// TIA Portal project "PaintMixingPlant" (V15)

(* hardware
DEVICE "S7-1200 station_1"  S7-1200 Station
   slot 0: "Rack_0"  S7-1200 Rack  Rack  V1.0
   slot 1: "PLC_1"  CPU 1214C AC/DC/Rly  6ES7 214-1BG40-0XB0  V4.2
DEVICE "PC-System_1"  SIMATIC PC station
   slot 0: "SIMATIC PC station"  Rail  SIMATIC PC-Station  V1.0
      slot 125: "Stationmanager"  Station_Manager  V6.0.4
   slot 1: "HMI_RT_1"  WinCC RT Professional  6AV2 105-0xxxx-xxxx  15.0.0.0
   slot 2: "IE general_1"  IE General  IE_CP  V8.2.0
*)

// ===== PLC "PLC_1"  CPU 1214C AC/DC/Rly =====

VAR_GLOBAL   // PLC tag table "Default tag table"
   "Mix1Tank1" AT %MW0 : Int;
   "Mix1Tank2" AT %MW2 : Int;
   "Mix1Tank3" AT %MW4 : Int;
   "Mix2Tank1" AT %MW6 : Int;
   "Mix2Tank2" AT %MW8 : Int;
   "Mix2Tank3" AT %MW10 : Int;
   "Mix3Tank1" AT %MW12 : Int;
   "Mix3Tank2" AT %MW14 : Int;
   "Mix3Tank3" AT %MW16 : Int;
   "InitM1T1" AT %MW18 : Int;
   "InitM1T2" AT %MW20 : Int;
   "InitM1T3" AT %MW22 : Int;
   "InitM2T1" AT %MW24 : Int;
   "InitM2T2" AT %MW26 : Int;
   "InitM2T3" AT %MW28 : Int;
   "InitM3T1" AT %MW30 : Int;
   "InitM3T2" AT %MW32 : Int;
   "InitM3T3" AT %MW34 : Int;
   "Tank1In" AT %MW36 : Int;
   "Tank1Out" AT %MW38 : Int;
   "Tank2In" AT %MW40 : Int;
   "Tank2Out" AT %MW42 : Int;
   "Tank3In" AT %MW44 : Int;
   "Tank3Out" AT %MW46 : Int;
   "Batch1In" AT %MW48 : Int;
   "Batch1Out" AT %MW50 : Int;
   "Batch2In" AT %MW52 : Int;
   "Batch2Out" AT %MW54 : Int;
   "Batch3In" AT %MW56 : Int;
   "Batch3Out" AT %MW58 : Int;
   "MixerIn" AT %MW60 : Int;
   "MixerOut" AT %MW62 : Int;
   "Start_Pb" AT %M64.0 : Bool;
   "Start_Trigger" AT %M64.1 : Bool;
   "Start" AT %M64.2 : Bool;
   "Stop_Pb" AT %M64.3 : Bool;
   "Stop_Trigger" AT %M64.4 : Bool;
   "InitStart" AT %M64.5 : Bool;
   "NextMix" AT %M64.6 : Bool;
   "ResetInd" AT %M64.7 : Bool;
   "Current_Mix" AT %MW66 : Int;
   "NumberOfMix1" AT %MW68 : Int;
   "Mix1Reset" AT %M65.0 : Bool;
   "NumberOfMix2" AT %MW70 : Int;
   "Mix2Reset" AT %M65.1 : Bool;
   "NumberOfMix3" AT %MW72 : Int;
   "Mix3Reset" AT %M65.2 : Bool;
   "Valve1_Mode" AT %M65.3 : Bool;
   "Valve2_Mode" AT %M65.4 : Bool;
   "Valve3_Mode" AT %M65.5 : Bool;
   "BatchValve1_Mode" AT %M65.6 : Bool;
   "BatchValve2_Mode" AT %M65.7 : Bool;
   "BatchValve3_Mode" AT %M74.0 : Bool;
   "MixerValve_mode" AT %M74.1 : Bool;
   "Tank1_MixingMode" AT %MW74 : Int;
   "Tank2_MixingMode" AT %MW76 : Int;
   "Tank3_MixingMode" AT %MW78 : Int;
   "Color_mode" AT %MW80 : Int;
   "Pump1" AT %M82.0 : Bool;
   "Pump2" AT %M82.1 : Bool;
   "Pump3" AT %M82.2 : Bool;
   "Pump1_Mode" AT %M82.3 : Bool;
   "Pump2_Mode" AT %M82.4 : Bool;
   "Pump3_Mode" AT %M82.5 : Bool;
   "Batch1_Done" AT %M82.6 : Bool;
   "Batch2_Done" AT %M82.7 : Bool;
   "Batch3_Done" AT %M83.0 : Bool;
   "Tank1_Valve" AT %M83.1 : Bool;
   "Tank2_Valve" AT %M83.2 : Bool;
   "Tank3_Valve" AT %M83.3 : Bool;
   "Batch1_Valve" AT %M83.4 : Bool;
   "Batch2_Valve" AT %M83.5 : Bool;
   "Batch3_Valve" AT %M83.6 : Bool;
   "Mixer" AT %M83.7 : Bool;
   "Mixer_Mode" AT %M84.0 : Bool;
   "MixerValve" AT %M84.1 : Bool;
   "Simple_Pulse" AT %M84.2 : Bool;
   "Stop" AT %M84.3 : Bool;
   "Tank4In" AT %MW86 : Int;
   "Tank4Out" AT %MW88 : Int;
   "Batch4In" AT %MW90 : Int;
   "Batch4Out" AT %MW92 : Int;
   "Mix1tank4" AT %MW94 : Int;
   "Mix2Tank4" AT %MW96 : Int;
   "Mix3Tank4" AT %MW98 : Int;
   "InitM1T4" AT %MW100 : Int;
   "InitM2T4" AT %MW102 : Int;
   "InitM3T4" AT %MW104 : Int;
   "Tank4_MixingMode" AT %MW106 : Int;
   "Batch4_Done" AT %M84.4 : Bool;
   "Pump4" AT %M84.5 : Bool;
   "Pump4_mode" AT %M84.6 : Bool;
   "Tank4_Valve" AT %M84.7 : Bool;
   "Batch4_Valve" AT %M85.0 : Bool;
   "Valve4_mode" AT %M85.1 : Bool;
   "BatchValve4_mode" AT %M85.2 : Bool;
   "Remaing_time" AT %MD108 : Time;
   "Remaing_time(1)" AT %MD112 : Time;
END_VAR

DATA_BLOCK "InitValues_DB"   // DB1
{ S7_Optimized_Access := 'TRUE' }
VERSION : 0.1
// stored: InstanceOfName InitValues
"InitValues"
BEGIN
END_DATA_BLOCK

DATA_BLOCK "I/OScaling_DB"   // DB2
{ S7_Optimized_Access := 'TRUE' }
VERSION : 0.1
// stored: InstanceOfName I/OScaling
"I/OScaling"
BEGIN
END_DATA_BLOCK

DATA_BLOCK "MixingRate_DB"   // DB7
{ S7_Optimized_Access := 'TRUE' }
VERSION : 0.1
// stored: InstanceOfName MixingRate
"MixingRate"
BEGIN
END_DATA_BLOCK

DATA_BLOCK "InitOperation_DB"   // DB8
{ S7_Optimized_Access := 'TRUE' }
VERSION : 0.1
// stored: InstanceOfName InitOperation
"InitOperation"
BEGIN
END_DATA_BLOCK

DATA_BLOCK "Pump_Operation_DB"   // DB20
{ S7_Optimized_Access := 'TRUE' }
VERSION : 0.1
// stored: InstanceOfName Pump_Operation
"Pump_Operation"
BEGIN
END_DATA_BLOCK

DATA_BLOCK "Tank_Valves_DB"   // DB21
{ S7_Optimized_Access := 'TRUE' }
VERSION : 0.1
// stored: InstanceOfName Tank_Valves
"Tank_Valves"
BEGIN
END_DATA_BLOCK

DATA_BLOCK "Batch_Valves_DB"   // DB28
{ S7_Optimized_Access := 'TRUE' }
VERSION : 0.1
// stored: InstanceOfName Batch_Valves
"Batch_Valves"
BEGIN
END_DATA_BLOCK

DATA_BLOCK "Mixer_Operation_DB"   // DB31
{ S7_Optimized_Access := 'TRUE' }
VERSION : 0.1
// stored: InstanceOfName Mixer_Operation
"Mixer_Operation"
BEGIN
END_DATA_BLOCK

// folder: System blocks/Program resources

DATA_BLOCK "Mixing_Order"   // DB3
{ S7_Optimized_Access := 'TRUE' }
AUTHOR : Simatic
FAMILY : IEC
NAME : CNTR
VERSION : 1.0
// stored: InstanceOfName IEC_COUNTER
"IEC_COUNTER"
BEGIN
END_DATA_BLOCK

DATA_BLOCK "Mix1Counter"   // DB4
{ S7_Optimized_Access := 'TRUE' }
AUTHOR : Simatic
FAMILY : IEC
NAME : CNTR
VERSION : 1.0
// stored: InstanceOfName IEC_COUNTER
"IEC_COUNTER"
BEGIN
END_DATA_BLOCK

DATA_BLOCK "Mix2Counter"   // DB5
{ S7_Optimized_Access := 'TRUE' }
AUTHOR : Simatic
FAMILY : IEC
NAME : CNTR
VERSION : 1.0
// stored: InstanceOfName IEC_COUNTER
"IEC_COUNTER"
BEGIN
END_DATA_BLOCK

DATA_BLOCK "Mix3Counter"   // DB6
{ S7_Optimized_Access := 'TRUE' }
AUTHOR : Simatic
FAMILY : IEC
NAME : CNTR
VERSION : 1.0
// stored: InstanceOfName IEC_COUNTER
"IEC_COUNTER"
BEGIN
END_DATA_BLOCK

DATA_BLOCK "IEC_Timer_0_DB"   // DB11
{ S7_Optimized_Access := 'TRUE' }
AUTHOR : Simatic
FAMILY : IEC
NAME : IEC_TMR
VERSION : 1.0
// stored: InstanceOfName IEC_TIMER
"IEC_TIMER"
BEGIN
END_DATA_BLOCK

DATA_BLOCK "IEC_Timer_0_DB_1"   // DB12
{ S7_Optimized_Access := 'TRUE' }
AUTHOR : Simatic
FAMILY : IEC
NAME : IEC_TMR
VERSION : 1.0
// stored: InstanceOfName IEC_TIMER
"IEC_TIMER"
BEGIN
END_DATA_BLOCK

DATA_BLOCK "IEC_Timer_0_DB_2"   // DB13
{ S7_Optimized_Access := 'TRUE' }
AUTHOR : Simatic
FAMILY : IEC
NAME : IEC_TMR
VERSION : 1.0
// stored: InstanceOfName IEC_TIMER
"IEC_TIMER"
BEGIN
END_DATA_BLOCK

DATA_BLOCK "IEC_Timer_0_DB_3"   // DB14
{ S7_Optimized_Access := 'TRUE' }
AUTHOR : Simatic
FAMILY : IEC
NAME : IEC_TMR
VERSION : 1.0
// stored: InstanceOfName IEC_TIMER
"IEC_TIMER"
BEGIN
END_DATA_BLOCK

DATA_BLOCK "IEC_Timer_0_DB_4"   // DB15
{ S7_Optimized_Access := 'TRUE' }
AUTHOR : Simatic
FAMILY : IEC
NAME : IEC_TMR
VERSION : 1.0
// stored: InstanceOfName IEC_TIMER
"IEC_TIMER"
BEGIN
END_DATA_BLOCK

DATA_BLOCK "IEC_Timer_0_DB_5"   // DB16
{ S7_Optimized_Access := 'TRUE' }
AUTHOR : Simatic
FAMILY : IEC
NAME : IEC_TMR
VERSION : 1.0
// stored: InstanceOfName IEC_TIMER
"IEC_TIMER"
BEGIN
END_DATA_BLOCK

DATA_BLOCK "IEC_Timer_0_DB_6"   // DB17
{ S7_Optimized_Access := 'TRUE' }
AUTHOR : Simatic
FAMILY : IEC
NAME : IEC_TMR
VERSION : 1.0
// stored: InstanceOfName IEC_TIMER
"IEC_TIMER"
BEGIN
END_DATA_BLOCK

DATA_BLOCK "IEC_Timer_0_DB_9"   // DB22
{ S7_Optimized_Access := 'TRUE' }
AUTHOR : Simatic
FAMILY : IEC
NAME : IEC_TMR
VERSION : 1.0
// stored: InstanceOfName IEC_TIMER
"IEC_TIMER"
BEGIN
END_DATA_BLOCK

DATA_BLOCK "IEC_Timer_0_DB_10"   // DB23
{ S7_Optimized_Access := 'TRUE' }
AUTHOR : Simatic
FAMILY : IEC
NAME : IEC_TMR
VERSION : 1.0
// stored: InstanceOfName IEC_TIMER
"IEC_TIMER"
BEGIN
END_DATA_BLOCK

DATA_BLOCK "IEC_Timer_0_DB_12"   // DB25
{ S7_Optimized_Access := 'TRUE' }
AUTHOR : Simatic
FAMILY : IEC
NAME : IEC_TMR
VERSION : 1.0
// stored: InstanceOfName IEC_TIMER
"IEC_TIMER"
BEGIN
END_DATA_BLOCK

DATA_BLOCK "IEC_Timer_0_DB_15"   // DB29
{ S7_Optimized_Access := 'TRUE' }
AUTHOR : Simatic
FAMILY : IEC
NAME : IEC_TMR
VERSION : 1.0
// stored: InstanceOfName IEC_TIMER
"IEC_TIMER"
BEGIN
END_DATA_BLOCK

DATA_BLOCK "IEC_Timer_0_DB_16"   // DB30
{ S7_Optimized_Access := 'TRUE' }
AUTHOR : Simatic
FAMILY : IEC
NAME : IEC_TMR
VERSION : 1.0
// stored: InstanceOfName IEC_TIMER
"IEC_TIMER"
BEGIN
END_DATA_BLOCK

DATA_BLOCK "IEC_Timer_0_DB_14"   // DB45
{ S7_Optimized_Access := 'TRUE' }
AUTHOR : Simatic
FAMILY : IEC
NAME : IEC_TMR
VERSION : 1.0
// stored: InstanceOfName IEC_TIMER
"IEC_TIMER"
BEGIN
END_DATA_BLOCK

DATA_BLOCK "IEC_Timer_0_DB_17"   // DB46
{ S7_Optimized_Access := 'TRUE' }
AUTHOR : Simatic
FAMILY : IEC
NAME : IEC_TMR
VERSION : 1.0
// stored: InstanceOfName IEC_TIMER
"IEC_TIMER"
BEGIN
END_DATA_BLOCK

DATA_BLOCK "IEC_Timer_0_DB_18"   // DB47
{ S7_Optimized_Access := 'TRUE' }
AUTHOR : Simatic
FAMILY : IEC
NAME : IEC_TMR
VERSION : 1.0
// stored: InstanceOfName IEC_TIMER
"IEC_TIMER"
BEGIN
END_DATA_BLOCK

DATA_BLOCK "IEC_Timer_0_DB_19"   // DB48
{ S7_Optimized_Access := 'TRUE' }
AUTHOR : Simatic
FAMILY : IEC
NAME : IEC_TMR
VERSION : 1.0
// stored: InstanceOfName IEC_TIMER
"IEC_TIMER"
BEGIN
END_DATA_BLOCK

DATA_BLOCK "IEC_Timer_0_DB_20"   // DB51
{ S7_Optimized_Access := 'TRUE' }
AUTHOR : Simatic
FAMILY : IEC
NAME : IEC_TMR
VERSION : 1.0
// stored: InstanceOfName IEC_TIMER
"IEC_TIMER"
BEGIN
END_DATA_BLOCK

DATA_BLOCK "IEC_Timer_0_DB_21"   // DB52
{ S7_Optimized_Access := 'TRUE' }
AUTHOR : Simatic
FAMILY : IEC
NAME : IEC_TMR
VERSION : 1.0
// stored: InstanceOfName IEC_TIMER
"IEC_TIMER"
BEGIN
END_DATA_BLOCK

// folder: (top level)

FUNCTION_BLOCK "InitValues"   // FB1, FBD
{ S7_Optimized_Access := 'TRUE' }
VERSION : 0.1
BEGIN

REGION Network 1
   // Tank Values For Mix1
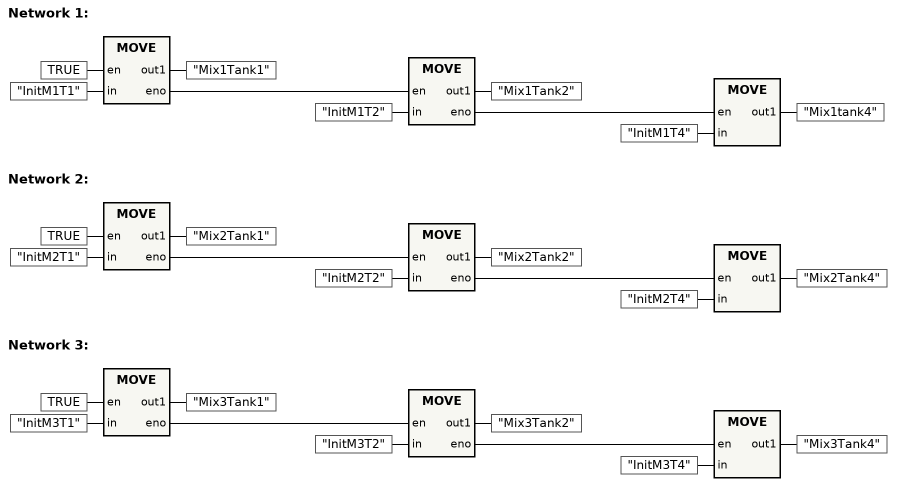
   IF TRUE THEN
       "Mix1Tank1" := "InitM1T1";
       "Mix1Tank2" := "InitM1T2";
       "Mix1tank4" := "InitM1T4";
   END_IF;
END_REGION

REGION Network 2
   // Tank Values For Mix2
   IF TRUE THEN
       "Mix2Tank1" := "InitM2T1";
       "Mix2Tank2" := "InitM2T2";
       "Mix2Tank4" := "InitM2T4";
   END_IF;
END_REGION

REGION Network 3
   // Tank Values For Mix3
   IF TRUE THEN
       "Mix3Tank1" := "InitM3T1";
       "Mix3Tank2" := "InitM3T2";
       "Mix3Tank4" := "InitM3T4";
   END_IF;
END_REGION
END_FUNCTION_BLOCK

FUNCTION_BLOCK "I/OScaling"   // FB2, FBD
{ S7_Optimized_Access := 'TRUE' }
VERSION : 0.1
BEGIN

REGION Network 1
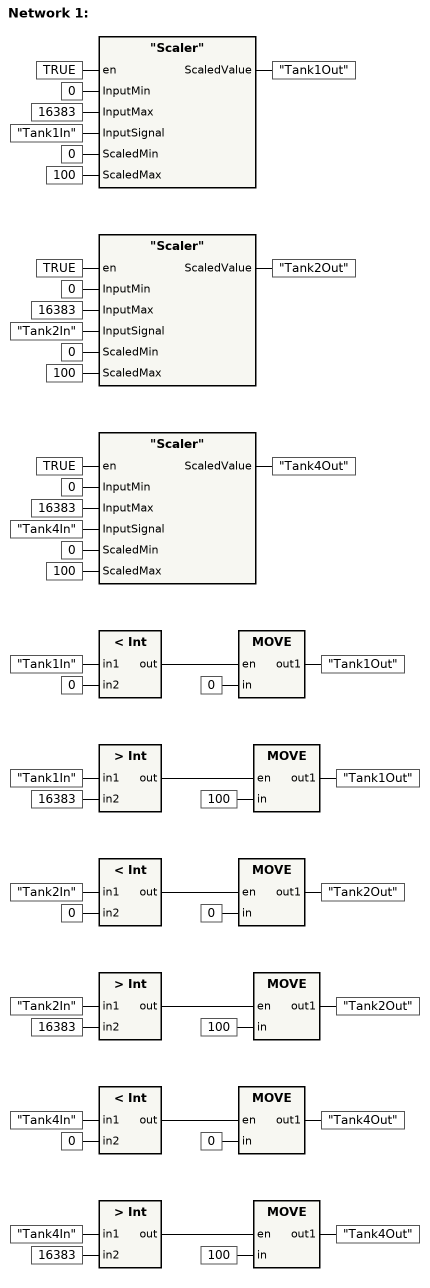
   IF TRUE THEN
       "Scaler"(InputMin := 0,
                InputMax := 16383,
                InputSignal := "Tank1In",
                ScaledMin := 0,
                ScaledMax := 100,
                ScaledValue => "Tank1Out");
       "Scaler"(InputMin := 0,
                InputMax := 16383,
                InputSignal := "Tank2In",
                ScaledMin := 0,
                ScaledMax := 100,
                ScaledValue => "Tank2Out");
       "Scaler"(InputMin := 0,
                InputMax := 16383,
                InputSignal := "Tank4In",
                ScaledMin := 0,
                ScaledMax := 100,
                ScaledValue => "Tank4Out");
   END_IF;
   IF "Tank1In" < 0 THEN "Tank1Out" := 0; END_IF;
   IF "Tank1In" > 16383 THEN "Tank1Out" := 100; END_IF;
   IF "Tank2In" < 0 THEN "Tank2Out" := 0; END_IF;
   IF "Tank2In" > 16383 THEN "Tank2Out" := 100; END_IF;
   IF "Tank4In" < 0 THEN "Tank4Out" := 0; END_IF;
   IF "Tank4In" > 16383 THEN "Tank4Out" := 100; END_IF;
END_REGION

REGION Network 2
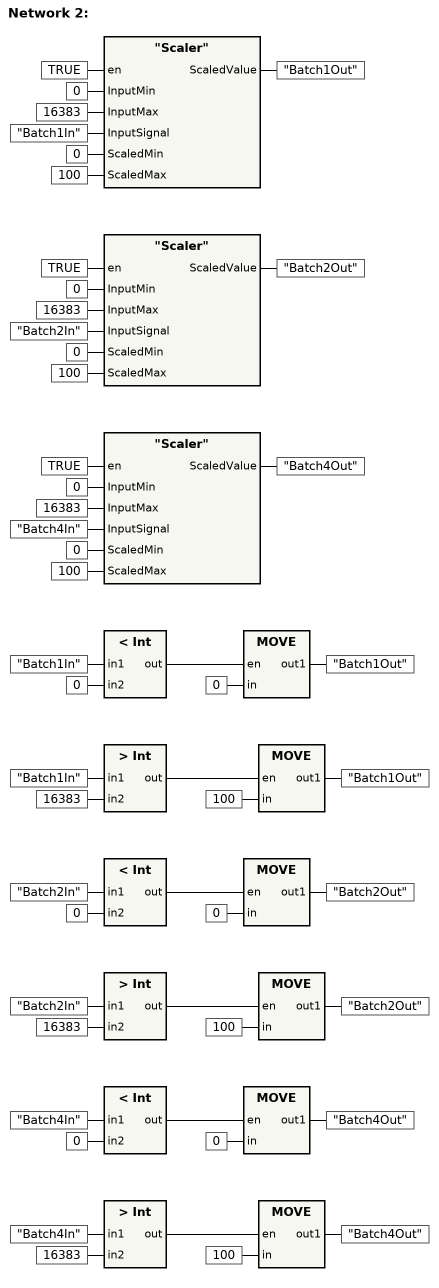
   IF TRUE THEN
       "Scaler"(InputMin := 0,
                InputMax := 16383,
                InputSignal := "Batch1In",
                ScaledMin := 0,
                ScaledMax := 100,
                ScaledValue => "Batch1Out");
       "Scaler"(InputMin := 0,
                InputMax := 16383,
                InputSignal := "Batch2In",
                ScaledMin := 0,
                ScaledMax := 100,
                ScaledValue => "Batch2Out");
       "Scaler"(InputMin := 0,
                InputMax := 16383,
                InputSignal := "Batch4In",
                ScaledMin := 0,
                ScaledMax := 100,
                ScaledValue => "Batch4Out");
   END_IF;
   IF "Batch1In" < 0 THEN "Batch1Out" := 0; END_IF;
   IF "Batch1In" > 16383 THEN "Batch1Out" := 100; END_IF;
   IF "Batch2In" < 0 THEN "Batch2Out" := 0; END_IF;
   IF "Batch2In" > 16383 THEN "Batch2Out" := 100; END_IF;
   IF "Batch4In" < 0 THEN "Batch4Out" := 0; END_IF;
   IF "Batch4In" > 16383 THEN "Batch4Out" := 100; END_IF;
END_REGION

REGION Network 3
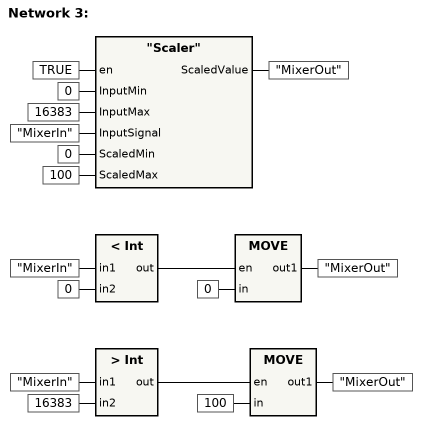
   IF TRUE THEN
       "Scaler"(InputMin := 0,
                InputMax := 16383,
                InputSignal := "MixerIn",
                ScaledMin := 0,
                ScaledMax := 100,
                ScaledValue => "MixerOut");
   END_IF;
   IF "MixerIn" < 0 THEN "MixerOut" := 0; END_IF;
   IF "MixerIn" > 16383 THEN "MixerOut" := 100; END_IF;
END_REGION
END_FUNCTION_BLOCK

FUNCTION_BLOCK "InitOperation"   // FB3, LAD
{ S7_Optimized_Access := 'TRUE' }
VERSION : 0.1
   VAR
      ons1 : Bool;
      ons2 : Bool;
      ResetONS : Bool;
   END_VAR
   VAR_TEMP   // added for the SCL form of the ladder/FBD networks
      _w1 : Bool;
      _w2 : Bool;
   END_VAR
BEGIN

REGION Network 1
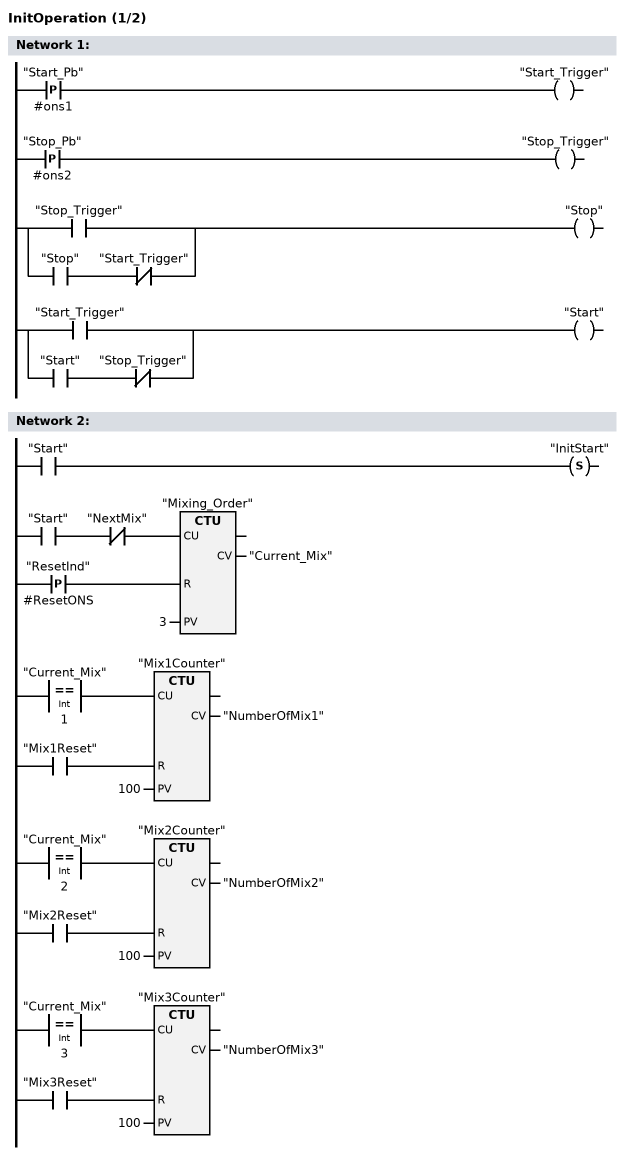
   RUNG wire#powerrail
      P_Contact(operand := "Start_Pb", bit := #ons1)
      Coil( "Start_Trigger" )
   END_RUNG
   RUNG wire#powerrail
      P_Contact(operand := "Stop_Pb", bit := #ons2)
      Coil( "Stop_Trigger" )
   END_RUNG
   RUNG wire#powerrail
      Contact( "Stop_Trigger" )
      wire#w1
      Coil( "Stop" )
   END_RUNG
   RUNG wire#powerrail
      Contact( "Stop" )
      I_Contact( "Start_Trigger" )
   END_RUNG wire#w1
   RUNG wire#powerrail
      Contact( "Start_Trigger" )
      wire#w2
      Coil( "Start" )
   END_RUNG
   RUNG wire#powerrail
      Contact( "Start" )
      I_Contact( "Stop_Trigger" )
   END_RUNG wire#w2
   // the same network as SCL:
   #_w1 := "Start_Pb" AND NOT #ons1;   // rising edge of "Start_Pb"
   #ons1 := "Start_Pb";
   "Start_Trigger" := #_w1;
   #_w2 := "Stop_Pb" AND NOT #ons2;   // rising edge of "Stop_Pb"
   #ons2 := "Stop_Pb";
   "Stop_Trigger" := #_w2;
   "Stop" := "Stop_Trigger" OR ("Stop" AND NOT "Start_Trigger");
   "Start" := "Start_Trigger" OR ("Start" AND NOT "Stop_Trigger");
END_REGION

REGION Network 2
   IF "Start" THEN "InitStart" := TRUE; END_IF;
   #_w1 := "ResetInd" AND NOT #ResetONS;   // rising edge of "ResetInd"
   #ResetONS := "ResetInd";
   "Mixing_Order".CTU(CU := "Start" AND NOT "NextMix", R := #_w1, PV := 3, CV => "Current_Mix");
   "Mix1Counter".CTU(CU := "Current_Mix" = 1, R := "Mix1Reset", PV := 100, CV => "NumberOfMix1");
   "Mix2Counter".CTU(CU := "Current_Mix" = 2, R := "Mix2Reset", PV := 100, CV => "NumberOfMix2");
   "Mix3Counter".CTU(CU := "Current_Mix" = 3, R := "Mix3Reset", PV := 100, CV => "NumberOfMix3");
END_REGION

REGION Network 3
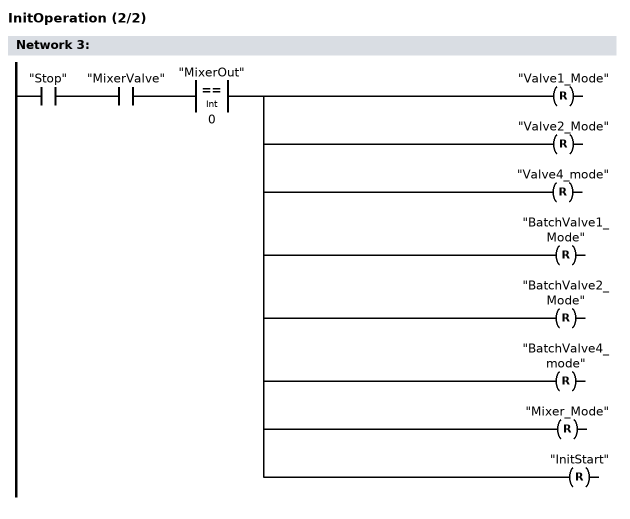
   RUNG wire#powerrail
      Contact( "Stop" )
      Contact( "MixerValve" )
      { S7_Templates := "SrcType := Int" } EQ_Contact(in1 := "MixerOut", in2 := 0)
      wire#w1
      R_Coil( "Valve1_Mode" )
   END_RUNG
   RUNG wire#w1
      R_Coil( "Valve2_Mode" )
   END_RUNG
   RUNG wire#w1
      R_Coil( "Valve4_mode" )
   END_RUNG
   RUNG wire#w1
      R_Coil( "BatchValve1_Mode" )
   END_RUNG
   RUNG wire#w1
      R_Coil( "BatchValve2_Mode" )
   END_RUNG
   RUNG wire#w1
      R_Coil( "BatchValve4_mode" )
   END_RUNG
   RUNG wire#w1
      R_Coil( "Mixer_Mode" )
   END_RUNG
   RUNG wire#w1
      R_Coil( "InitStart" )
   END_RUNG
   // the same network as SCL:
   IF "Stop" AND "MixerValve" AND ("MixerOut" = 0) THEN
       "Valve1_Mode" := FALSE;
       "Valve2_Mode" := FALSE;
       "Valve4_mode" := FALSE;
       "BatchValve1_Mode" := FALSE;
       "BatchValve2_Mode" := FALSE;
       "BatchValve4_mode" := FALSE;
       "Mixer_Mode" := FALSE;
       "InitStart" := FALSE;
   END_IF;
END_REGION
END_FUNCTION_BLOCK

FUNCTION_BLOCK "MixingRate"   // FB4, SCL
{ S7_Optimized_Access := 'TRUE' }
VERSION : 0.1
BEGIN
   IF "Current_Mix" = 1 THEN
       "Tank1_MixingMode" := "Mix1Tank1";
       "Tank2_MixingMode" := "Mix1Tank2";
       "Tank4_MixingMode" := "Mix1tank4";
       "Color_mode" := 1;
   END_IF;

   IF "Current_Mix" = 2 THEN
       "Tank1_MixingMode" := "Mix2Tank1";
       "Tank2_MixingMode" := "Mix2Tank2";
       "Tank4_MixingMode" := "Mix2Tank4";
       "Color_mode" := 2;
   END_IF;

   IF "Current_Mix" = 3 THEN
       "Tank1_MixingMode" := "Mix3Tank1";
       "Tank2_MixingMode" := "Mix3Tank2";
       "Tank4_MixingMode" := "Mix3Tank4";
       "Color_mode" := 3;
   END_IF;

   IF "Current_Mix" = 0 THEN
       "Tank1_MixingMode" := 1;
       "Tank2_MixingMode" := 1;
       "Tank4_MixingMode" := 1;
       "Color_mode" := 3;
   END_IF;
END_FUNCTION_BLOCK

FUNCTION_BLOCK "Pump_Operation"   // FB5, SCL
{ S7_Optimized_Access := 'TRUE' }
VERSION : 0.1
   VAR_TEMP
      Pump1_Start_Set : Bool;
      tv1 : Time;
      Pump1_Stop_Set : Bool;
      tv2 : Time;
      Pump1_Pumping : Bool;
      tv3 : Time;
      Pump2_Start_Set : Bool;
      tv4 : Time;
      Pump2_stop_Set : Bool;
      tv5 : Time;
      Pump2_Pumping : Bool;
      tv6 : Time;
      Pump3_Start_Set : Bool;
      tv7 : Time;
      Pump3_Stop_Set : Bool;
      tv8 : Time;
      Pump3_Pumping : Bool;
      tv9 : Time;
      Pump4_Start_Set : Bool;
      tv10 : Time;
      Pump4_Stop_Set : Bool;
      tv11 : Time;
      Pump4_pumping : Bool;
      tv12 : Time;
   END_VAR
BEGIN
   IF "Pump1_Mode" = 1 THEN

       "IEC_Timer_0_DB".TON(IN := TRUE,
                            PT := T#500ms,
                            Q => #Pump1_Start_Set,
                            ET => #tv1);
   END_IF;

   IF "Pump1_Mode" = 0 THEN

       "IEC_Timer_0_DB_1".TON(IN := TRUE,
                              PT := T#500ms,
                              Q => #Pump1_Stop_Set,
                              ET => #tv2);
   END_IF;

   IF #Pump1_Start_Set THEN
       "Pump1" := 1;
       "IEC_Timer_0_DB_2".TON(IN := TRUE,
                              PT := T#200ms,
                              Q => #Pump1_Pumping,
                              ET => #tv3);
       IF #Pump1_Pumping THEN
           RESET_TIMER("IEC_Timer_0_DB_2");
           "Tank1In" := "Tank1In" + 50;
       END_IF;
   END_IF;

   IF #Pump1_Stop_Set THEN
       "Pump1" := 0;
   END_IF;

   IF "Pump2_Mode" = 1 THEN

       "IEC_Timer_0_DB_3".TON(IN := TRUE,
                              PT := T#500ms,
                              Q => #Pump2_Start_Set,
                              ET => #tv4);
   END_IF;

   IF "Pump2_Mode" = 0 THEN

       "IEC_Timer_0_DB_4".TON(IN := TRUE,
                              PT := T#500ms,
                              Q => #Pump2_stop_Set,
                              ET => #tv5);
   END_IF;

   IF #Pump2_Start_Set THEN
       "Pump2" := 1;
       "IEC_Timer_0_DB_5".TON(IN := TRUE,
                              PT := T#200ms,
                              Q => #Pump2_Pumping,
                              ET => #tv6);
       IF #Pump1_Pumping THEN
           RESET_TIMER("IEC_Timer_0_DB_5");
           "Tank2In" := "Tank2In" + 50;
       END_IF;
   END_IF;

   IF #Pump2_stop_Set THEN
       "Pump2" := 0;
   END_IF;

   IF "Pump4_mode" = 1 THEN

       "IEC_Timer_0_DB_17".TON(IN := TRUE,
                               PT := T#500ms,
                               Q => #Pump4_Start_Set,
                               ET => #tv10);
   END_IF;

   IF "Pump4_mode" = 0 THEN

       "IEC_Timer_0_DB_18".TON(IN := TRUE,
                               PT := T#500ms,
                               Q => #Pump4_Stop_Set,
                               ET => #tv11);
   END_IF;

   IF #Pump4_Start_Set THEN
       "Pump4" := 1;
       "IEC_Timer_0_DB_19".TON(IN := TRUE,
                               PT := T#200ms,
                               Q => #Pump4_pumping,
                               ET => #tv12);
       IF #Pump4_pumping THEN
           RESET_TIMER("IEC_Timer_0_DB_19");
           "Tank4In" := "Tank4In" + 50;
       END_IF;
   END_IF;

   IF #Pump4_Stop_Set THEN
       "Pump4" := 0;
   END_IF;

   IF "Tank1Out" < 30 THEN
       "Pump1_Mode" := 1;
   ELSIF "Tank1Out" > 80 THEN
       "Pump1_Mode" := 0;
   END_IF;

   IF "Tank2Out" < 30 THEN
       "Pump2_Mode" := 1;
   ELSIF "Tank2Out" > 80 THEN
       "Pump2_Mode" := 0;
   END_IF;

   IF "Tank4Out" < 30 THEN
       "Pump4_mode" := 1;
   ELSIF "Tank4Out" > 80 THEN
       "Pump4_mode" := 0;
   END_IF;
END_FUNCTION_BLOCK

FUNCTION_BLOCK "Tank_Valves"   // FB6, SCL
{ S7_Optimized_Access := 'TRUE' }
VERSION : 0.1
   VAR
      Mode2Set : Bool;
      Mode3Set : Bool;
      Mode1Reset : Bool;
      Mode1Set : Bool;
      Mode2Reset : Bool;
      Mode3Reset : Bool;
      Done1 : Bool;
      Done2 : Bool;
      Done3 : Bool;
      Done4 : Bool;
      Mode4Set : Bool;
      Mode4Reset : Bool;
   END_VAR
BEGIN
   IF "InitStart" AND "Tank1_MixingMode" = 1 THEN
       "R_TRIG_DB_11"(CLK:=TRUE,
                      Q=>#Done1);
       IF #Done1 THEN
           "Batch1_Done" := 1;
       END_IF;
   END_IF;

   IF "InitStart" AND "Tank2_MixingMode" = 1 THEN
       "R_TRIG_DB_12"(CLK := TRUE,
                      Q => #Done2);
       IF #Done2 THEN
           "Batch2_Done" := 1;
       END_IF;
   END_IF;

   IF "InitStart" AND "Tank4_MixingMode" = 1 THEN
       "R_TRIG_DB_15"(CLK := TRUE,
                      Q => #Done4);
       IF #Done4 THEN
           "Batch4_Done" := 1;
       END_IF;
   END_IF;


   IF ("Tank1_MixingMode" = 3 AND "InitStart" AND "Tank1Out" > 30) OR ("Tank1_MixingMode" = 2 AND
       "InitStart" AND "Tank1Out" > 30) THEN
       "R_TRIG_DB"(CLK := TRUE,
                   Q => #Mode1Set);
       IF #Mode1Set THEN
           "Valve1_Mode" := 1;
       END_IF;
   END_IF;

   IF ("Tank1_MixingMode" = 3 AND "Tank1Out" > 30 AND "Batch1Out" >=100) OR ("Tank1_MixingMode" = 2 AND
       "Tank1Out" > 30 AND "Batch1Out" >=50) THEN
       "R_TRIG_DB_3"(CLK := TRUE,
                     Q => #Mode1Reset);
       IF #Mode1Reset THEN
           "Valve1_Mode" := 0;
           "BatchValve1_Mode" := 1;
       END_IF;
   END_IF;

   IF ("Tank2_MixingMode" = 3 AND "InitStart" AND "Tank2Out" > 30) OR ("Tank2_MixingMode" = 2 AND
       "InitStart" AND "Tank2Out" > 30) THEN
       "R_TRIG_DB_1"(CLK := TRUE,
                     Q => #Mode2Set);
       IF #Mode2Set THEN
           "Valve2_Mode" := 1;
       END_IF;
   END_IF;

   IF ("Tank2_MixingMode" = 3 AND "Tank2Out" > 30 AND "Batch2Out" >=100) OR ("Tank2_MixingMode" = 2 AND
       "Tank2Out" > 30 AND "Batch2Out" >=50) THEN
       "R_TRIG_DB_4"(CLK:=TRUE,
                     Q=>#Mode2Reset);
       IF #Mode2Reset THEN
           "Valve2_Mode" := 0;
           "BatchValve2_Mode" := 1;
       END_IF;
   END_IF;

   IF ("Tank4_MixingMode" = 3 AND "InitStart" AND "Tank4Out" > 30) OR ("Tank4_MixingMode" = 2 AND
       "InitStart" AND "Tank4Out" > 30) THEN
       "R_TRIG_DB_16"(CLK := TRUE,
                      Q => #Mode4Set);
       IF #Mode4Set THEN
           "Valve4_mode" := 1;
       END_IF;
   END_IF;

   IF ("Tank4_MixingMode" = 3 AND "Tank4Out" > 30 AND "Batch4Out" >= 100) OR ("Tank4_MixingMode" = 2 AND
       "Tank4Out" > 30 AND "Batch4Out" >= 50) THEN
       "R_TRIG_DB_17"(CLK := TRUE,
                      Q => #Mode4Reset);
       IF #Mode4Reset THEN
           "Valve4_mode" := 0;
           "BatchValve4_mode" := 1;
       END_IF;
   END_IF;
END_FUNCTION_BLOCK

FUNCTION_BLOCK "Batch_Valves"   // FB7, SCL
{ S7_Optimized_Access := 'TRUE' }
VERSION : 0.1
   VAR
      Batch1ModeSet : Bool;
      Batch2ModeSet : Bool;
      Batch3ModeSet : Bool;
      Batch4ModeSet : Bool;
   END_VAR
   VAR_TEMP
      Valve1Set : Bool;
      t1 : Time;
      Valve2Set : Bool;
      t2 : Time;
      Valve3Set : Bool;
      t3 : Time;
      Batch1Set : Bool;
      t4 : Time;
      Batch2Set : Bool;
      t5 : Time;
      Batch3Set : Bool;
      t6 : Time;
      Valve4Set : Bool;
      t7 : Time;
      Batch4Set : Bool;
      t8 : Time;
   END_VAR
BEGIN
   IF "Valve1_Mode" THEN
       "Tank1_Valve" := 1;
       "IEC_Timer_0_DB_9".TON(IN := TRUE,
                              PT := T#200ms,
                              Q => #Valve1Set,
                              ET => #t1);
       IF #Valve1Set THEN
           RESET_TIMER("IEC_Timer_0_DB_9");
           "Batch1In" := "Batch1In" + 100;
           "Tank1In" := "Tank1In" - 30;
       END_IF;
   END_IF;

   IF NOT "Valve1_Mode" THEN
       "Tank1_Valve" := 0;
   END_IF;

   IF "Valve2_Mode" THEN
       "Tank2_Valve" := 1;
       "IEC_Timer_0_DB_10".TON(IN:=TRUE,
                               PT:=T#200ms,
                               Q=>#Valve2Set,
                               ET=>#t2);
       IF #Valve2Set THEN
           RESET_TIMER("IEC_Timer_0_DB_10");
           "Batch2In" := "Batch2In" + 100;
           "Tank2In" := "Tank2In" - 30;
       END_IF;
   END_IF;

   IF NOT "Valve2_Mode" THEN
       "Tank2_Valve" := 0;
   END_IF;

   IF "Valve4_mode" THEN
       "Tank4_Valve" := 1;
       "IEC_Timer_0_DB_20".TON(IN := TRUE,
                               PT := T#200ms,
                               Q => #Valve4Set,
                               ET => #t7);
       IF #Valve4Set THEN
           RESET_TIMER("IEC_Timer_0_DB_20");
           "Batch4In" := "Batch4In" + 100;
           "Tank4In" := "Tank4In" - 30;
       END_IF;
   END_IF;


   IF NOT "Valve4_mode" THEN
       "Tank4_Valve" := 0;
   END_IF;

   IF "BatchValve1_Mode" THEN
       "Batch1_Valve" := 1;
       "IEC_Timer_0_DB_12".TON(IN := TRUE,
                               PT := T#200ms,
                               Q => #Batch1Set,
                               ET => #t4);
       IF #Batch1Set THEN
           RESET_TIMER("IEC_Timer_0_DB_12");
           "Batch1In" := "Batch1In" - 100;
           "MixerIn" := "MixerIn" + 30;
       END_IF;
       IF "Batch1Out" <= 0 THEN
           "R_TRIG_DB_6"(CLK := TRUE,
                         Q => #Batch1ModeSet);
           IF #Batch1ModeSet THEN
               "R_TRIG_DB_6"(CLK := FALSE);
               "BatchValve1_Mode" := 0;
               "Batch1_Valve" := 0;
               "Batch1_Done" := 1;
           END_IF;
       END_IF;
   END_IF;


   IF "BatchValve2_Mode" THEN
       "Batch2_Valve" := 1;
       "IEC_Timer_0_DB_14".TON(IN := TRUE,
                               PT := T#200ms,
                               Q => #Batch2Set,
                               ET => #t5);
       IF #Batch2Set THEN
           RESET_TIMER("IEC_Timer_0_DB_14");
           "Batch2In" := "Batch2In" - 100;
           "MixerIn" := "MixerIn" + 30;
       END_IF;
       IF "Batch2Out" <= 0 THEN
           "R_TRIG_DB_7"(CLK := TRUE,
                         Q => #Batch2ModeSet);
           IF #Batch2ModeSet THEN
               "R_TRIG_DB_7"(CLK := FALSE);
               "BatchValve2_Mode" := 0;
               "Batch2_Valve" := 0;
               "Batch2_Done" := 1;
           END_IF;
       END_IF;
   END_IF;

   IF "BatchValve4_mode" THEN
       "Batch4_Valve" := 1;
       "IEC_Timer_0_DB_21".TON(IN := TRUE,
                               PT := T#200ms,
                               Q => #Batch4Set,
                               ET => #t8);
       IF #Batch4Set THEN
           RESET_TIMER("IEC_Timer_0_DB_21");
           "Batch4In" := "Batch4In" - 100;
           "MixerIn" := "MixerIn" + 30;
       END_IF;
       IF "Batch4Out" <= 0 THEN
           "R_TRIG_DB_18"(CLK := TRUE,
                          Q => #Batch4ModeSet);
           IF #Batch4ModeSet THEN
               "R_TRIG_DB_18"(CLK := FALSE);
               "BatchValve4_mode" := 0;
               "Batch4_Valve" := 0;
               "Batch4_Done" := 1;
           END_IF;
       END_IF;
   END_IF;
END_FUNCTION_BLOCK

FUNCTION_BLOCK "Mixer_Operation"   // FB8, SCL
{ S7_Optimized_Access := 'TRUE' }
VERSION : 0.1
   VAR
      ResetPulse : Bool;
      NextPulse : Bool;
      NextOne : Bool;
      ResetBit : Bool;
   END_VAR
   VAR_TEMP
      MixingDone : Bool;
      t7 : Time;
      MixingPulse : Bool;
      t8 : Time;
      NextBit : Bool;
      t9 : Time;
   END_VAR
BEGIN
   IF "Batch1_Done" AND "Batch2_Done" AND "Batch4_Done" AND "Current_Mix"<>0 THEN
       "Mixer_Mode" := 1;
   END_IF;

   IF "Mixer_Mode" AND "Current_Mix" <> 0 THEN
       "Mixer" := 1;
       "IEC_Timer_0_DB_15".TON(IN := TRUE,
                               PT := T#5s,
                               Q => #MixingDone,
                               ET => #t7);
       IF #MixingDone THEN
           RESET_TIMER("IEC_Timer_0_DB_15");

           "Mixer" := 0;
           "Batch1_Done" := 0;
           "Batch2_Done" := 0;
           "Batch4_Done" := 0;
           "Mixer_Mode" := 0;
           "MixerValve_mode" := 1;
       END_IF;
   END_IF;


   IF "InitStart" AND "Current_Mix" = 0 THEN
       "Mixer_Mode" := 0;
       "Batch1_Done" := 0;
       "Batch2_Done" := 0;
       "Batch4_Done" := 0;
       "NextMix" := 1;
       "IEC_Timer_0_DB_6".TON(IN:=TRUE,
                              PT:=T#100ms,
                              Q=>#NextBit,
                              ET=>#t9);
       IF #NextBit THEN
           RESET_TIMER("IEC_Timer_0_DB_6");
           "NextMix" := 0;
       END_IF;

   END_IF;


   IF "MixerValve_mode" THEN
       "R_TRIG_DB_14"(CLK:=TRUE,
                      Q=>#NextOne);
       IF #NextOne THEN
           "R_TRIG_DB_14"(CLK := FALSE);
           "NextMix" := 1;
           "MixerValve" := 1;
       END_IF;
   END_IF;


   IF "MixerValve" THEN

       "IEC_Timer_0_DB_16".TON(IN := TRUE,
                               PT := T#200ms,
                               Q => #MixingPulse,
                               ET => #t8);
       IF #MixingPulse THEN
           RESET_TIMER("IEC_Timer_0_DB_16");
           "MixerIn" := "MixerIn" - 200;
       END_IF;
   END_IF;


   IF "Current_Mix" = 3 AND "MixerValve" AND "MixerOut"=0 THEN
       "R_TRIG_DB_9"(CLK := TRUE,
                     Q => #ResetPulse);
       IF #ResetPulse THEN
           "R_TRIG_DB_9"(CLK := FALSE);
           "ResetInd" := 1;
       END_IF;
   END_IF;

   IF "Current_Mix" = 3 AND "MixerValve" AND "MixerOut" > 10 THEN
       "R_TRIG_DB_5"(CLK:=TRUE,
                     Q=>#ResetBit);
       IF #ResetBit THEN
           "R_TRIG_DB_5"(CLK := FALSE);
           "ResetInd" := 0;
       END_IF;
   END_IF;


   IF "MixerValve"  AND "MixerOut" = 0 THEN
       "R_TRIG_DB_10"(CLK := TRUE,
                      Q => #NextPulse);
       IF #NextPulse THEN
           "R_TRIG_DB_10"(CLK := FALSE);
           "MixerValve_mode" := 0;
           "MixerValve" := 0;
           "NextMix" := 0;
           "R_TRIG_DB_11"(CLK := FALSE);
           "R_TRIG_DB_12"(CLK := FALSE);
           "R_TRIG_DB_15"(CLK := FALSE);
           "R_TRIG_DB"(CLK := FALSE);
           "R_TRIG_DB_3"(CLK := FALSE);
           "R_TRIG_DB_1"(CLK := FALSE);
           "R_TRIG_DB_4"(CLK := FALSE);
           "R_TRIG_DB_16"(CLK := FALSE);
           "R_TRIG_DB_17"(CLK := FALSE);
       END_IF;
   END_IF;
END_FUNCTION_BLOCK

FUNCTION "Scaler" : Void   // FC1, LAD
{ S7_Optimized_Access := 'TRUE' }
VERSION : 0.1
   VAR_INPUT
      InputMin : Int;
      InputMax : Int;
      InputSignal : Int;
      ScaledMin : Int;
      ScaledMax : Int;
   END_VAR
   VAR_OUTPUT
      ScaledValue : Int;
   END_VAR
   VAR_TEMP
      tv : Real;
   END_VAR
BEGIN

REGION Network 1
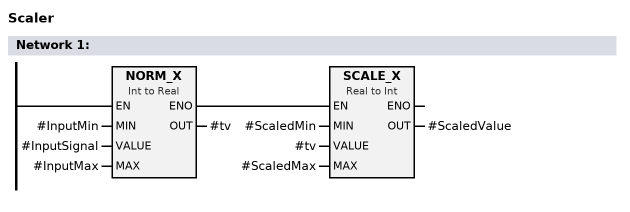
   RUNG wire#powerrail
      { S7_Templates := "[SrcType := Int, DestType := Real]" } Normalize(min := #InputMin, value := #InputSignal, max := #InputMax, out => #tv)
      { S7_Templates := "[SrcType := Real, DestType := Int]" } Scale(min := #ScaledMin, value := #tv, max := #ScaledMax, out => #ScaledValue)
   END_RUNG
   // the same network as SCL:
   #tv := NORM_X(MIN := #InputMin, VALUE := #InputSignal, MAX := #InputMax);
   #ScaledValue := SCALE_X(MIN := #ScaledMin, VALUE := #tv, MAX := #ScaledMax);
END_REGION
END_FUNCTION

ORGANIZATION_BLOCK "Main"   // OB1, LAD, ProgramCycle
TITLE = "Main Program Sweep (Cycle)"
{ S7_Optimized_Access := 'TRUE' }
VERSION : 0.1
   VAR_INPUT
      Initial_Call : Bool;   // Initial call of this OB
      Remanence : Bool;   // =True, if remanent data are available
   END_VAR
   VAR_TEMP   // added for the SCL form of the ladder/FBD networks
      _w1 : Bool;
   END_VAR
BEGIN

REGION Network 1
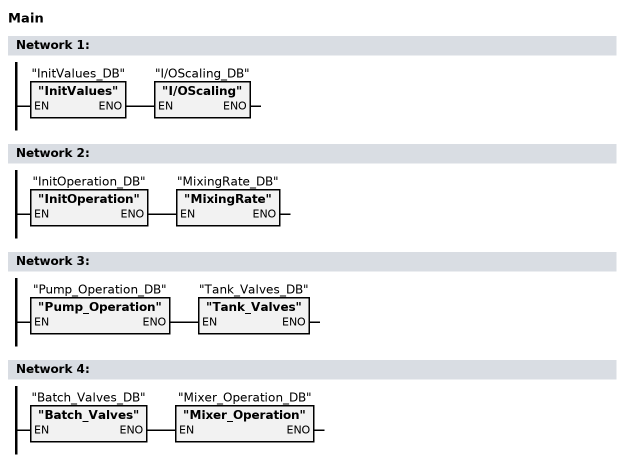
   RUNG wire#powerrail
      "InitValues_DB"()
      "I/OScaling_DB"()
   END_RUNG
   // the same network as SCL:
   "InitValues_DB"(ENO => #_w1);   // "InitValues"
   IF #_w1 THEN
       "I/OScaling_DB"();   // "I/OScaling"
   END_IF;
END_REGION

REGION Network 2
   RUNG wire#powerrail
      "InitOperation_DB"()
      "MixingRate_DB"()
   END_RUNG
   // the same network as SCL:
   "InitOperation_DB"(ENO => #_w1);   // "InitOperation"
   IF #_w1 THEN
       "MixingRate_DB"();   // "MixingRate"
   END_IF;
END_REGION

REGION Network 3
   RUNG wire#powerrail
      "Pump_Operation_DB"()
      "Tank_Valves_DB"()
   END_RUNG
   // the same network as SCL:
   "Pump_Operation_DB"(ENO => #_w1);   // "Pump_Operation"
   IF #_w1 THEN
       "Tank_Valves_DB"();   // "Tank_Valves"
   END_IF;
END_REGION

REGION Network 4
   RUNG wire#powerrail
      "Batch_Valves_DB"()
      "Mixer_Operation_DB"()
   END_RUNG
   // the same network as SCL:
   "Batch_Valves_DB"(ENO => #_w1);   // "Batch_Valves"
   IF #_w1 THEN
       "Mixer_Operation_DB"();   // "Mixer_Operation"
   END_IF;
END_REGION
END_ORGANIZATION_BLOCK

(* ===== HMI "HMI_RT_1" =====
system functions are stored by id; their names below are inferred from use
connection "HMI_Connection_1": S71200_TCP_IP, SCADA_S7_1200

HMI tags "Default tag table"
   "Tank1Out" : Int = PLC Tank1Out AT %MW38, 500 ms
   "Tank2Out" : Int = PLC Tank2Out AT %MW42, 500 ms
   "Tank3Out" : Int = PLC Tank3Out AT %MW46, 500 ms
   "Pump1_Mode" : Bool = PLC Pump1_Mode AT %M82.3, 500 ms
   "Pump2_Mode" : Bool = PLC Pump2_Mode AT %M82.4, 500 ms
   "Batch1Out" : Int = PLC Batch1Out AT %MW50, 500 ms
   "Batch2Out" : Int = PLC Batch2Out AT %MW54, 500 ms
   "Batch3Out" : Int = PLC Batch3Out AT %MW58, 500 ms
   "Tank1Valve" : Bool = PLC Tank1_Valve AT %M83.1, 500 ms
   "Tank2Valve" : Bool = PLC Tank2_Valve AT %M83.2, 500 ms
   "Tank3Valve" : Bool = PLC Tank3_Valve AT %M83.3, 500 ms
   "Batch1Valve" : Bool = PLC Batch1_Valve AT %M83.4, 500 ms
   "Batch2Valve" : Bool = PLC Batch2_Valve AT %M83.5, 500 ms
   "Batch3Valve" : Bool = PLC Batch3_Valve AT %M83.6, 500 ms
   "MixerOut" : Int = PLC MixerOut AT %MW62, 500 ms
   "Pump1" : Bool = PLC Pump1 AT %M82.0, 500 ms
   "Pump2" : Bool = PLC Pump2 AT %M82.1, 500 ms
   "Start_Pb" : Bool = PLC Start_Pb AT %M64.0, 500 ms
   "Stop_Pb" : Bool = PLC Stop_Pb AT %M64.3, 500 ms
   "InitM1T1" : Int = PLC InitM1T1 AT %MW18, 500 ms
   "InitM1T2" : Int = PLC InitM1T2 AT %MW20, 500 ms
   "InitM1T3" : Int = PLC InitM1T3 AT %MW22, 500 ms
   "InitM2T1" : Int = PLC InitM2T1 AT %MW24, 500 ms
   "InitM2T2" : Int = PLC InitM2T2 AT %MW26, 500 ms
   "InitM2T3" : Int = PLC InitM2T3 AT %MW28, 500 ms
   "InitM3T1" : Int = PLC InitM3T1 AT %MW30, 500 ms
   "InitM3T2" : Int = PLC InitM3T2 AT %MW32, 500 ms
   "InitM3T3" : Int = PLC InitM3T3 AT %MW34, 500 ms
   "Start" : Bool = PLC Start AT %M64.2, 500 ms
   "Stop" : Bool = PLC Stop AT %M84.3, 500 ms
   "InitM1T4" : Int = PLC InitM1T4 AT %MW100, 500 ms
   "InitM2T4" : Int = PLC InitM2T4 AT %MW102, 500 ms
   "InitM3T4" : Int = PLC InitM3T4 AT %MW104, 500 ms
   "Batch4Out" : Int = PLC Batch4Out AT %MW92, 500 ms
   "Batch4Valve" : Bool = PLC Batch4_Valve AT %M85.0, 500 ms
   "Pump4" : Bool = PLC Pump4 AT %M84.5, 500 ms
   "Pump4_Mode" : Bool = PLC Pump4_mode AT %M84.6, 500 ms
   "Tank4Out" : Int = PLC Tank4Out AT %MW88, 500 ms
   "Tank4Valve" : Bool = PLC Tank4_Valve AT %M84.7, 500 ms
   "MixerMode" : Bool = PLC Mixer_Mode AT %M84.0, 500 ms
   "MixerValve" : Bool = PLC MixerValve AT %M84.1, 500 ms
   "Mixer" : Bool = PLC Mixer AT %M83.7, 500 ms
   "NumberOfMix1" : Int = PLC NumberOfMix1 AT %MW68, 500 ms
   "NumberOfMix2" : Int = PLC NumberOfMix2 AT %MW70, 500 ms
   "NumberOfMix3" : Int = PLC NumberOfMix3 AT %MW72, 500 ms

graphic list "MixerBlade": 1 'MixerBlades'

recipe "ColorMix": Mix1Tank1 <- "InitM1T1", Mix1Tank2 <- "InitM1T2", Mix2Tank1 <- "InitM2T1", Mix2Tank2 <- "InitM2T2", Mix3Tank1 <- "InitM3T1", Mix3Tank2 <- "InitM3T2", Mix1Tank4 <- "InitM1T4", Mix2Tank4 <- "InitM2T4", Mix3tank4 <- "InitM3T4"

screen "Main_Schematic" 900x600
   Bar "Bar_7" at 378,421 size 193x105; MinimumValue 0; MaximumValue 100
      ProcessValue <- "MixerOut"
   TubePolyline "Pipe_5" at 289,511 size 98x0
   TubePolyline "Pipe_24" at 543,377 size 0x44
   TubePolyline "Pipe_25" at 497,355 size 34x1
   TubePolyline "Pipe_21" at 425,359 size 21x0
   TubePolyline "Pipe_18" at 412,237 size 0x111
   TubePolyline "Pipe_16" at 412,178 size 0x89
   TubePolyline "Pipe_17" at 682,188 size 0x65
   TubePolyline "Pipe_20" at 694,354 size 22x1
   TubePolyline "Pipe_19" at 682,238 size 0x104
   TubePolyline "Pipe_4" at 681,367 size 37x1
   TubePolyline "Pipe_22" at 670,382 size 0x51
   TubePolyline "Pipe_11" at 670,425 size 0x69
   TubePolyline "Pipe_23" at 564,508 size 95x0
   TubePolyline "Pipe_12" at 275,425 size 0x73
   TubePolyline "Pipe_13" at 275,368 size 0x61
   TubePolyline "Pipe_3" at 230,356 size 33x1
   TubePolyline "Pipe_6" at 161,359 size 19x1
   TubePolyline "Pipe_15" at 147,191 size 0x59
   TubePolyline "Pipe_9" at 623,176 size 65x0
   TubePolyline "Pipe_10" at 356,185 size 61x0
   TubePolyline "Pipe_8" at 92,187 size 54x1
   TextField "Text field_1" at 344,14 size 212x28; Text 'MAIN SCHEMATIC'
   Group "Group" at 137,78 size 138x136
   Group "Group_1" at 405,78 size 138x136
   Group "Group_2" at 673,78 size 138x136
   Bar "Bar_1" at 147,98 size 118x105; MinimumValue 0; MaximumValue 100
      ProcessValue <- "Tank1Out"
   Bar "Bar_2" at 415,98 size 118x105; MinimumValue 0; MaximumValue 100
      ProcessValue <- "Tank2Out"
   Bar "Bar_3" at 685,98 size 118x105; MinimumValue 0; MaximumValue 100
      ProcessValue <- "Tank4Out"
   GraphicView "Graphic view_1" at 57,170 size 49x35; Picture "Graphic_2"
      Visibility <- "Pump1"
   GraphicView "Graphic view_2" at 57,169 size 50x36; Picture "Graphic_3"
      Visibility <- "Pump1"
   GraphicView "Graphic view_3" at 597,159 size 49x35; Picture "Graphic_2"
      Visibility <- "Pump4"
   GraphicView "Graphic view_4" at 319,169 size 49x35; Picture "Graphic_2"
      Visibility <- "Pump2"
   GraphicView "Graphic view_5" at 319,167 size 49x38; Picture "Graphic_3"
      Visibility <- "Pump2"
   GraphicView "Graphic view_6" at 598,158 size 48x36; Picture "Graphic_3"
      Visibility <- "Pump4"
   Group "Group_3" at 171,259 size 67x123
   Bar "Bar_4" at 181,279 size 47x92; MinimumValue 0; MaximumValue 100
      ProcessValue <- "Batch1Out"
   Group "Group_4" at 439,263 size 68x120
   Bar "Bar_5" at 449,283 size 48x89; MinimumValue 0; MaximumValue 100
      ProcessValue <- "Batch2Out"
   Group "Group_5" at 709,261 size 68x121
   Bar "Bar_6" at 721,281 size 48x90; MinimumValue 0; MaximumValue 100
      ProcessValue <- "Batch4Out"
   GraphicView "Graphic view_29" at 659,410 size 37x33; Picture "Graphic_8"
      Visibility <- "Batch4Valve"
   GraphicView "Graphic view_30" at 659,410 size 38x33; Picture "Graphic_9"
      Visibility <- "Batch4Valve"
   GraphicView "Graphic view_33" at 263,405 size 34x31; Picture "Graphic_8"
      Visibility <- "Batch1Valve"
   GraphicView "Graphic view_34" at 263,405 size 35x31; Picture "Graphic_9"
      Visibility <- "Batch1Valve"
   TubePolyline "Pipe_1" at 60,300 size 0x0
   TubePolyline "Pipe_2" at 34,269 size 0x0
   TubePolyline "Pipe_7" at 543,366 size 0x13
   TubePolyline "Pipe_14" at 147,238 size 0x109
   TubeArcObject "Pipe elbow_1" at 142,344 size 23x20
   TubeArcObject "Pipe elbow_2" at 655,490 size 20x23
   TubeArcObject "Pipe elbow_3" at 257,351 size 23x20
   TubeArcObject "Pipe elbow_4" at 665,363 size 20x25
   GraphicView "Graphic view_10" at 137,226 size 35x31; Picture "Graphic_8"
      Visibility <- "Tank1Valve"
   GraphicView "Graphic view_11" at 137,226 size 35x32; Picture "Graphic_9"
      Visibility <- "Tank1Valve"
   GraphicView "Graphic view_14" at 403,228 size 33x33; Picture "Graphic_8"
      Visibility <- "Tank2Valve"
   GraphicView "Graphic view_13" at 403,228 size 34x33; Picture "Graphic_9"
      Visibility <- "Tank2Valve"
   GraphicView "Graphic view_15" at 672,232 size 35x33; Picture "Graphic_8"
      Visibility <- "Tank4Valve"
   GraphicView "Graphic view_12" at 670,233 size 37x33; Picture "Graphic_9"
      Visibility <- "Tank4Valve"
   TubeArcObject "Pipe elbow_5" at 677,341 size 20x19
   TubeArcObject "Pipe elbow_6" at 407,344 size 23x20
   TubeArcObject "Pipe elbow_7" at 270,495 size 23x21
   TubeArcObject "Pipe elbow_8" at 525,350 size 23x20
   GraphicView "Graphic view_31" at 531,370 size 40x33; Picture "Graphic_8"
      Visibility <- "Batch2Valve"
   GraphicView "Graphic view_32" at 531,370 size 39x33; Picture "Graphic_9"
      Visibility <- "Batch2Valve"
   Button "Button_1" at 806,561 size 80x31; TextOff 'EXIT'
      on Click: StopRuntime(0)
   Button "Button_2" at 12,561 size 80x30; TextOff 'START'
      on PressLeft: SetBit("Start_Pb")
      on ReleaseLeft: ResetBit("Start_Pb")
      Appearance <- "Start"
   Button "Button_3" at 98,561 size 80x30; TextOff 'STOP'
      on PressLeft: SetBit("Stop_Pb")
      on ReleaseLeft: ResetBit("Stop_Pb")
      Appearance <- "Start"
   Button "Button_4" at 589,563 size 111x32; TextOff 'MIX CONFIG'
      on Click: ActivateScreen("Mixing_Configuration", 0)
   Group "Group_6" at 368,401 size 213x136
   TextField "Text field_2" at 177,63 size 51x18; Text 'TANK1'
   TextField "Text field_3" at 446,63 size 51x18; Text 'TANK2'
   TextField "Text field_4" at 709,63 size 51x18; Text 'TANK3'
   TextField "Text field_5" at 181,237 size 60x18; Text 'BATCH1'
   TextField "Text field_6" at 449,237 size 60x18; Text 'BATCH2'
   TextField "Text field_7" at 713,237 size 60x18; Text 'BATCH3'
   TextField "Text field_8" at 326,388 size 91x18; Text 'MIXERTANK'
   IOField "I/O field_1" at 272,211 size 34x18; FormatPattern 999
      ProcessValue <- "Tank1Out"
   TextField "Text field_9" at 308,211 size 15x18; Text '%'
   IOField "I/O field_2" at 591,480 size 34x18; FormatPattern 999
      ProcessValue <- "MixerOut"
   IOField "I/O field_3" at 785,329 size 34x18; FormatPattern 999
      ProcessValue <- "Batch4Out"
   IOField "I/O field_4" at 514,329 size 34x18; FormatPattern 999
      ProcessValue <- "Batch2Out"
   IOField "I/O field_5" at 247,329 size 34x18; FormatPattern 999
      ProcessValue <- "Batch1Out"
   IOField "I/O field_6" at 811,211 size 34x18; FormatPattern 999
      ProcessValue <- "Tank4Out"
   IOField "I/O field_7" at 542,211 size 34x18; FormatPattern 999
      ProcessValue <- "Tank2Out"
   TextField "Text field_10" at 627,480 size 15x18; Text '%'
   TextField "Text field_11" at 821,328 size 15x18; Text '%'
   TextField "Text field_12" at 556,328 size 15x18; Text '%'
   TextField "Text field_13" at 285,328 size 15x18; Text '%'
   TextField "Text field_14" at 849,211 size 15x18; Text '%'
   TextField "Text field_15" at 580,211 size 15x18; Text '%'
   GraphicView "Graphic view_7" at 368,447 size 215x81; Picture "MixerBlades"
      Visibility <- "Mixer"
   TextField "Text field_16" at 449,447 size 50x18; Text 'MIXER'
      Visibility <- "Mixer"
   GraphicView "Graphic view_8" at 439,503 size 70x58; Picture "Valve"
      Visibility <- "MixerValve"
   Button "Button_5" at 708,562 size 89x32; TextOff 'STATUS'
      on Click: ActivateScreen("Current_Status", 0)

screen "Mixing_Configuration" 900x600
   TextField "Text field_1" at 298,14 size 304x28; Text 'MIXING CONFIGURATION'
   UserArchiveControl "Recipe view_1" at 11,62 size 879x324; DataSource "ColorMix"
   TextField "Text field_2" at 287,416 size 323x23; Text 'ColorMix1: Color1, Color2, Color3'
   TextField "Text field_3" at 287,450 size 323x23; Text 'ColorMix1: Color4, Color5, Color6'
   TextField "Text field_4" at 287,484 size 323x23; Text 'ColorMix1: Color7, Color8, Color9'
   Button "Button_1" at 710,562 size 81x32; TextOff 'MAIN'
      on Click: ActivateScreen("Main_Schematic", 0)
   Button "Button_4" at 799,562 size 89x32; TextOff 'STATUS'
      on Click: ActivateScreen("Current_Status", 0)

screen "Current_Status" 900x600
   TextField "Text field_1" at 344,14 size 210x28; Text 'CURRENT STATUS'
   Button "Button_4" at 776,560 size 111x32; TextOff 'MIX CONFIG'
      on Click: ActivateScreen("Mixing_Configuration", 0)
   Button "Button_1" at 689,560 size 81x32; TextOff 'MAIN'
      on Click: ActivateScreen("Main_Schematic", 0)
   IOField "I/O field_1" at 218,267 size 111x61; FormatPattern 999
      ProcessValue <- "NumberOfMix1"
   IOField "I/O field_2" at 395,267 size 111x64; FormatPattern 999
      ProcessValue <- "NumberOfMix2"
   IOField "I/O field_3" at 572,267 size 111x63; FormatPattern 999
      ProcessValue <- "NumberOfMix3"
   TextField "Text field_2" at 234,209 size 433x33; Text 'THE NUMBER OF CURRENT MIX'
   TextField "Text field_3" at 571,364 size 112x33; Text 'COLOR3'
   TextField "Text field_4" at 393,364 size 112x33; Text 'COLOR2'
   TextField "Text field_5" at 222,364 size 106x33; Text 'CLOLR1'
*)